(* IEC 61131-3 sources: Industry-PLC-LLM/data/PLCBEAD_repo/PLCBEAD_PLCEmbed-main/PLC-BEAD/Source/GEB/SENSOR_INT, 1 file *)

(* ---- SENSOR_INT.ST ---- *)
FUNCTION SENSOR_INT:REAL

	VAR_INPUT
		VOLTAGE :	REAL;
		CURRENT :	REAL;
		RP :	REAL;
		_RS :	REAL;
	END_VAR

	VAR
		RG :	REAL;
	END_VAR

	IF current <> 0.0 THEN
		RG := voltage / current;
		SENSOR_INT := RP * ( RG - _RS) / ( RP + _RS - RG);
	END_IF;

END_FUNCTION

PROGRAM program0

	VAR
		VOLTAGE :	REAL;
		CURRENT :	REAL;
		RP :	REAL;
		_RS :	REAL;
		CEIL5_OUT : REAL;
	END_VAR

	CEIL5_OUT := SENSOR_INT(VOLTAGE, CURRENT, RP, _RS);

END_PROGRAM
